(* PLC project SafeLOGIC-1, BrAutomation SafeDESIGNER  4.3.2.11 *)
(* stored: companyURL http://www.br-automation.com, creationDateTime Thu May 17 17:30:16 2018 *)

PROGRAM ScaleSAFEDINT

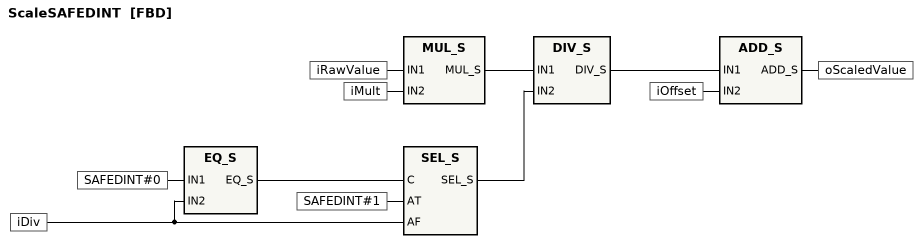
(* FBD diagram, written out as Structured Text *)
oScaledValue := ADD_S(DIV_S(MUL_S(iRawValue, iMult), SEL_S(EQ_S(SAFEDINT#0, iDiv), SAFEDINT#1, iDiv)), iOffset);
END_PROGRAM
